Universal Robots URScript: command04.urscript

def returnHomeLinear():
  movel([0.3665191429,-2.234021443,-1.658062789,-0.8028514559,1.570796327,1.919862177], a=3.0, v=0.8)
  movel([0.03490658504,-2.225294796,-1.675516082,-0.7941248097,1.570796327,1.588249619], a=3.0, v=0.8)
  movel([-1.570796327,-1.570796327,-1.570796327,-1.570796327,1.570796327,0], a=3.0, v=0.8)
end
